// TIA Portal V15.1 export
// export: Created 2024-05-17T05:38:39.5671025Z, ExportSetting WithDefaults, DisplayName Totally Integrated Automation Portal, DisplayVersion V15.1 Update 5, DisplayName TIA Portal Openness, DisplayVersion V15.1 Update 5, DisplayName SINAMICS Startdrive Advanced, DisplayVersion V15.1, DisplayName G130, G150, S120, S150, SINAMICS MV, S210, DisplayVersion V15.1, DisplayName G110M, G120, G120C, G120D, G120P, DisplayVersion V15.1, DisplayName STEP 7 Professional, DisplayVersion V15.1 Update 5, DisplayName STEP 7 Safety, DisplayVersion V15.1, DisplayName WinCC Professional, DisplayVersion V15.1 Update 5, DisplayName SIMATIC Visualization Architect, DisplayVersion V15.1
FUNCTION_BLOCK "LGBBodyPitch"   // FB6657, FBD
TITLE = LRoller2W2S-MoviFitFCPN / LGBBodyPitch
{ S7_Optimized_Access := 'TRUE' }
AUTHOR : Imtech
FAMILY : Transport
VERSION : 0.1
// =============================================================================
// This module is used in Applications when a roller one way two speed equipped 
// with SEW MOVIFIT-FC is needed. The roller can support single body tranport and 
// simultanious transport. The roller is equipped with a standard sensor setting, 
// one stop High Speed and one at the front for dual speed transport. The 
// roller uses standard handshaking signals to accomplish an infeed transfer 
// with the previous transport system and an outfeed with the next transport 
// system.
// The roller will support automatic Mode and manual Mode according specific 
// guidelines.
// The outfeed will be master over the infeed.
// Alarm "body not in Position" is also generated.
// All Alarms coming from sub-functions, TrfIn, TrfOut & LMotor2W2S-MoviFitFCPN or 
// from 
// local Alarm are summarized to give also the global Alarm A, B, C & D to 
// upper level.
// =============================================================================
// ============================================================================
// The BodyPitch function is a local FB to be used in blowing lines transport 
// functions to handle the pitchtime between bodys.
// ============================================================================
// stored: AutoNumber false, IsIECCheckEnabled false, IsRetainMemResEnabled false, MemoryReserve 100, SetENOAutomatically False, UDAEnableTagReadback false
   VAR_INPUT
      I_PrevBodyPresentDet { ExternalAccessible := 'False'; ExternalVisible := 'False'; ExternalWritable := 'False'} : Bool;   // Previous position body present
      I_PitchDet { ExternalAccessible := 'False'; ExternalVisible := 'False'; ExternalWritable := 'False'} : Bool;   // Pitch position present
      I_ConveyorMode { ExternalAccessible := 'False'; ExternalVisible := 'False'; ExternalWritable := 'False'} : Bool;
      I_ActualPitchVal { ExternalAccessible := 'False'; ExternalVisible := 'False'; ExternalWritable := 'False'} : Int;   // Encoder pitch value in cm
      I_SkidFrontToPitchVal { ExternalAccessible := 'False'; ExternalVisible := 'False'; ExternalWritable := 'False'} : Int;   // Encoder skidfront to pitch1 value in cm
      I_PrevTransferTm { ExternalAccessible := 'False'; ExternalVisible := 'False'; ExternalWritable := 'False'} : Bool;   // Transfer previous active
      I_MotorForwardActive { ExternalAccessible := 'False'; ExternalVisible := 'False'; ExternalWritable := 'False'} : Bool;   // Motor is moving forward
      C_ConvMovFwdTime { ExternalAccessible := 'False'; ExternalVisible := 'False'; ExternalWritable := 'False'} : Time;   // Conveyor move forward time
   END_VAR
   VAR_OUTPUT
      O_BodyPitchOK { ExternalAccessible := 'False'; ExternalVisible := 'False'; ExternalWritable := 'False'} : Bool;   // Body Pitch ok
      O_ResetActualPitchVal { ExternalAccessible := 'False'; ExternalVisible := 'False'; ExternalWritable := 'False'} : Bool;   // Reset actual pitch value
      O_ResetSkidFrontToPitVal { ExternalAccessible := 'False'; ExternalVisible := 'False'; ExternalWritable := 'False'} : Bool;   // Reset skidFront to Pitch value
      O_AlarmABCondition { ExternalAccessible := 'False'; ExternalVisible := 'False'; ExternalWritable := 'False'} : Bool;   // Alarm AB Condition
      O_AlarmA { ExternalAccessible := 'False'; ExternalVisible := 'False'; ExternalWritable := 'False'} : Bool;   // Alarm A
      O_AlarmB { ExternalAccessible := 'False'; ExternalVisible := 'False'; ExternalWritable := 'False'} : Bool;   // Alarm B
      O_AlarmC { ExternalAccessible := 'False'; ExternalVisible := 'False'; ExternalWritable := 'False'} : Bool;   // Alarm C
      O_AlarmD { ExternalAccessible := 'False'; ExternalVisible := 'False'; ExternalWritable := 'False'} : Bool;   // Alarm D
   END_VAR
   VAR_IN_OUT
      IO_Modes : "Modes";   // Modes
      H_HMI : "H_HMI";   // Animation
      H_GBBodyPitch : "H_GBBodyPitch";   // Animation
   END_VAR
   VAR
      BodyPitchOK { ExternalAccessible := 'False'; ExternalVisible := 'False'; ExternalWritable := 'False'} : Bool;   // Body pitch is ok
      PitchControlWithEncoder { ExternalAccessible := 'False'; ExternalVisible := 'False'; ExternalWritable := 'False'} : Bool;   // Pitch control with encoder active
      PitchControlWithTimer { ExternalAccessible := 'False'; ExternalVisible := 'False'; ExternalWritable := 'False'} : Bool;   // Pitch control with timer active
      PitchTimeReached { ExternalAccessible := 'False'; ExternalVisible := 'False'; ExternalWritable := 'False'} : Bool;   // Pitch time is reached
      PitchDistanceReached { ExternalAccessible := 'False'; ExternalVisible := 'False'; ExternalWritable := 'False'} : Bool;   // Pitch distance is reached
      PresenceBody { ExternalAccessible := 'False'; ExternalVisible := 'False'; ExternalWritable := 'False'} : Bool;   // Body present at begin of conveyor
      AlarmA { ExternalAccessible := 'False'; ExternalVisible := 'False'; ExternalWritable := 'False'} : Bool;   // Alarm A
      AlarmB { ExternalAccessible := 'False'; ExternalVisible := 'False'; ExternalWritable := 'False'} : Bool;   // Alarm B
      AlarmC { ExternalAccessible := 'False'; ExternalVisible := 'False'; ExternalWritable := 'False'} : Bool;   // Alarm C
      AlarmD { ExternalAccessible := 'False'; ExternalVisible := 'False'; ExternalWritable := 'False'} : Bool;   // Alarm D
      AlarmABCondition { ExternalAccessible := 'False'; ExternalVisible := 'False'; ExternalWritable := 'False'} : Bool;   // Alarm AB Condition
      Edge { ExternalAccessible := 'False'; ExternalVisible := 'False'; ExternalWritable := 'False'} : Array[1..7] of Bool;   // Edge
      TimerConvMovForw { ExternalAccessible := 'False'; ExternalVisible := 'False'; ExternalWritable := 'False'} : TOF_TIME;   // Timer
      PitchTimer { ExternalAccessible := 'False'; ExternalVisible := 'False'; ExternalWritable := 'False'} : "LTimer";   // Pitch Timer
   END_VAR
   VAR_TEMP
      HMICMD : Struct   // Temp
         PitchControlWithTimerSel : Bool;   // Pitch control with timer selected
         PitchControlWithEncoderSel : Bool;   // Pitch control with encoder selected
         Spare2 : Bool;   // Spare
         Spare3 : Bool;   // Spare
         Spare4 : Bool;   // Spare
         Spare5 : Bool;   // Spare
         Spare6 : Bool;   // Spare
         Spare7 : Bool;   // Spare
         Spare8 : Bool;   // Spare
         Spare9 : Bool;   // Spare
         Spare10 : Bool;   // Spare
         Spare11 : Bool;   // Spare
         Spare12 : Bool;   // Spare
         Spare13 : Bool;   // Spare
         Spare14 : Bool;   // Spare
         Spare15 : Bool;   // Spare
         Spare16 : Bool;   // Spare
         Spare17 : Bool;   // Spare
         Spare18 : Bool;   // Spare
         Spare19 : Bool;   // Spare
         Spare20 : Bool;   // Spare
         Spare21 : Bool;   // Spare
         Spare22 : Bool;   // Spare
         Spare23 : Bool;   // Spare
         Spare24 : Bool;   // Spare
         Spare25 : Bool;   // Spare
         Spare26 : Bool;   // Spare
         Spare27 : Bool;   // Spare
         Spare28 : Bool;   // Spare
         Spare29 : Bool;   // Spare
         Spare30 : Bool;   // Spare
         Spare31 : Bool;   // Spare
      END_STRUCT;
      TempInt : Int;   // Temp
      TempDInt : DInt;   // Temp / Temp DInt
      TempReal : Real;   // Temp
   END_VAR
   VAR_TEMP   // added for the SCL form of the ladder/FBD networks
      _w1 : Bool;
      _w2 : Bool;
   END_VAR
BEGIN

REGION Network 1: **** 1 - Inputs **** HMI Commands
   // HMI Commands
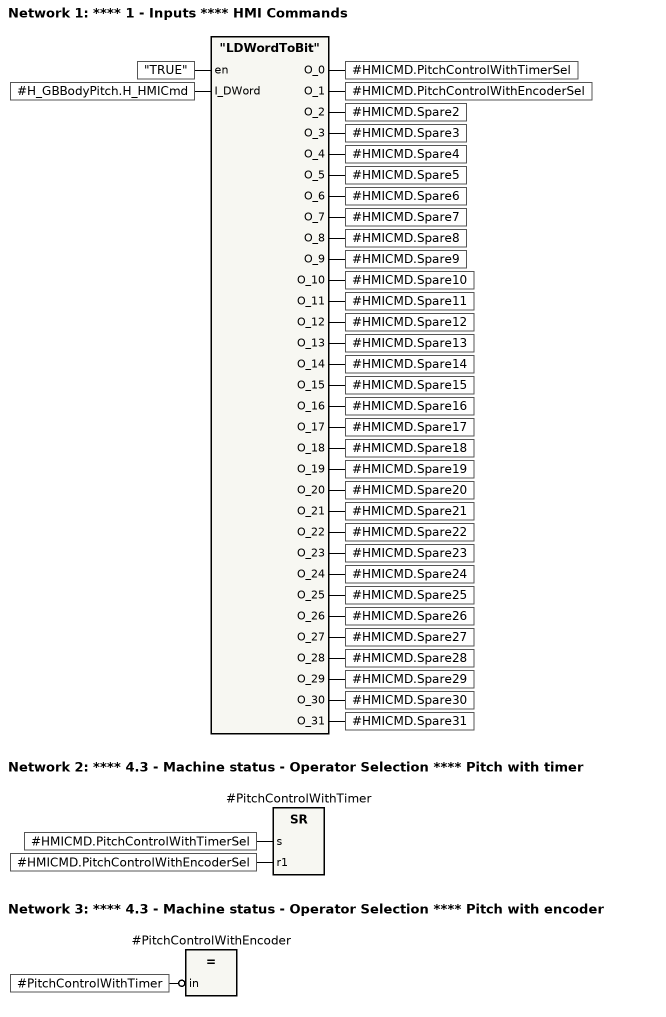
   IF "TRUE" THEN
       "LDWordToBit"(I_DWord := #H_GBBodyPitch.H_HMICmd,
                     O_0 => #HMICMD.PitchControlWithTimerSel,
                     O_1 => #HMICMD.PitchControlWithEncoderSel,
                     O_2 => #HMICMD.Spare2,
                     O_3 => #HMICMD.Spare3,
                     O_4 => #HMICMD.Spare4,
                     O_5 => #HMICMD.Spare5,
                     O_6 => #HMICMD.Spare6,
                     O_7 => #HMICMD.Spare7,
                     O_8 => #HMICMD.Spare8,
                     O_9 => #HMICMD.Spare9,
                     O_10 => #HMICMD.Spare10,
                     O_11 => #HMICMD.Spare11,
                     O_12 => #HMICMD.Spare12,
                     O_13 => #HMICMD.Spare13,
                     O_14 => #HMICMD.Spare14,
                     O_15 => #HMICMD.Spare15,
                     O_16 => #HMICMD.Spare16,
                     O_17 => #HMICMD.Spare17,
                     O_18 => #HMICMD.Spare18,
                     O_19 => #HMICMD.Spare19,
                     O_20 => #HMICMD.Spare20,
                     O_21 => #HMICMD.Spare21,
                     O_22 => #HMICMD.Spare22,
                     O_23 => #HMICMD.Spare23,
                     O_24 => #HMICMD.Spare24,
                     O_25 => #HMICMD.Spare25,
                     O_26 => #HMICMD.Spare26,
                     O_27 => #HMICMD.Spare27,
                     O_28 => #HMICMD.Spare28,
                     O_29 => #HMICMD.Spare29,
                     O_30 => #HMICMD.Spare30,
                     O_31 => #HMICMD.Spare31);
   END_IF;
END_REGION

REGION Network 2: **** 4.3 - Machine status - Operator Selection **** Pitch with timer
   IF #HMICMD.PitchControlWithTimerSel THEN
       #PitchControlWithTimer := TRUE;   // SR flip-flop
   END_IF;
   IF #HMICMD.PitchControlWithEncoderSel THEN #PitchControlWithTimer := FALSE; END_IF;
END_REGION

REGION Network 3: **** 4.3 - Machine status - Operator Selection **** Pitch with encoder
   #PitchControlWithEncoder := NOT #PitchControlWithTimer;
END_REGION

REGION Network 4: **** 4.4 - Machine status - Calculated **** Logger skidfront - pitch sensor distance
   // Simple logger for skidfront - pitch sensor distance
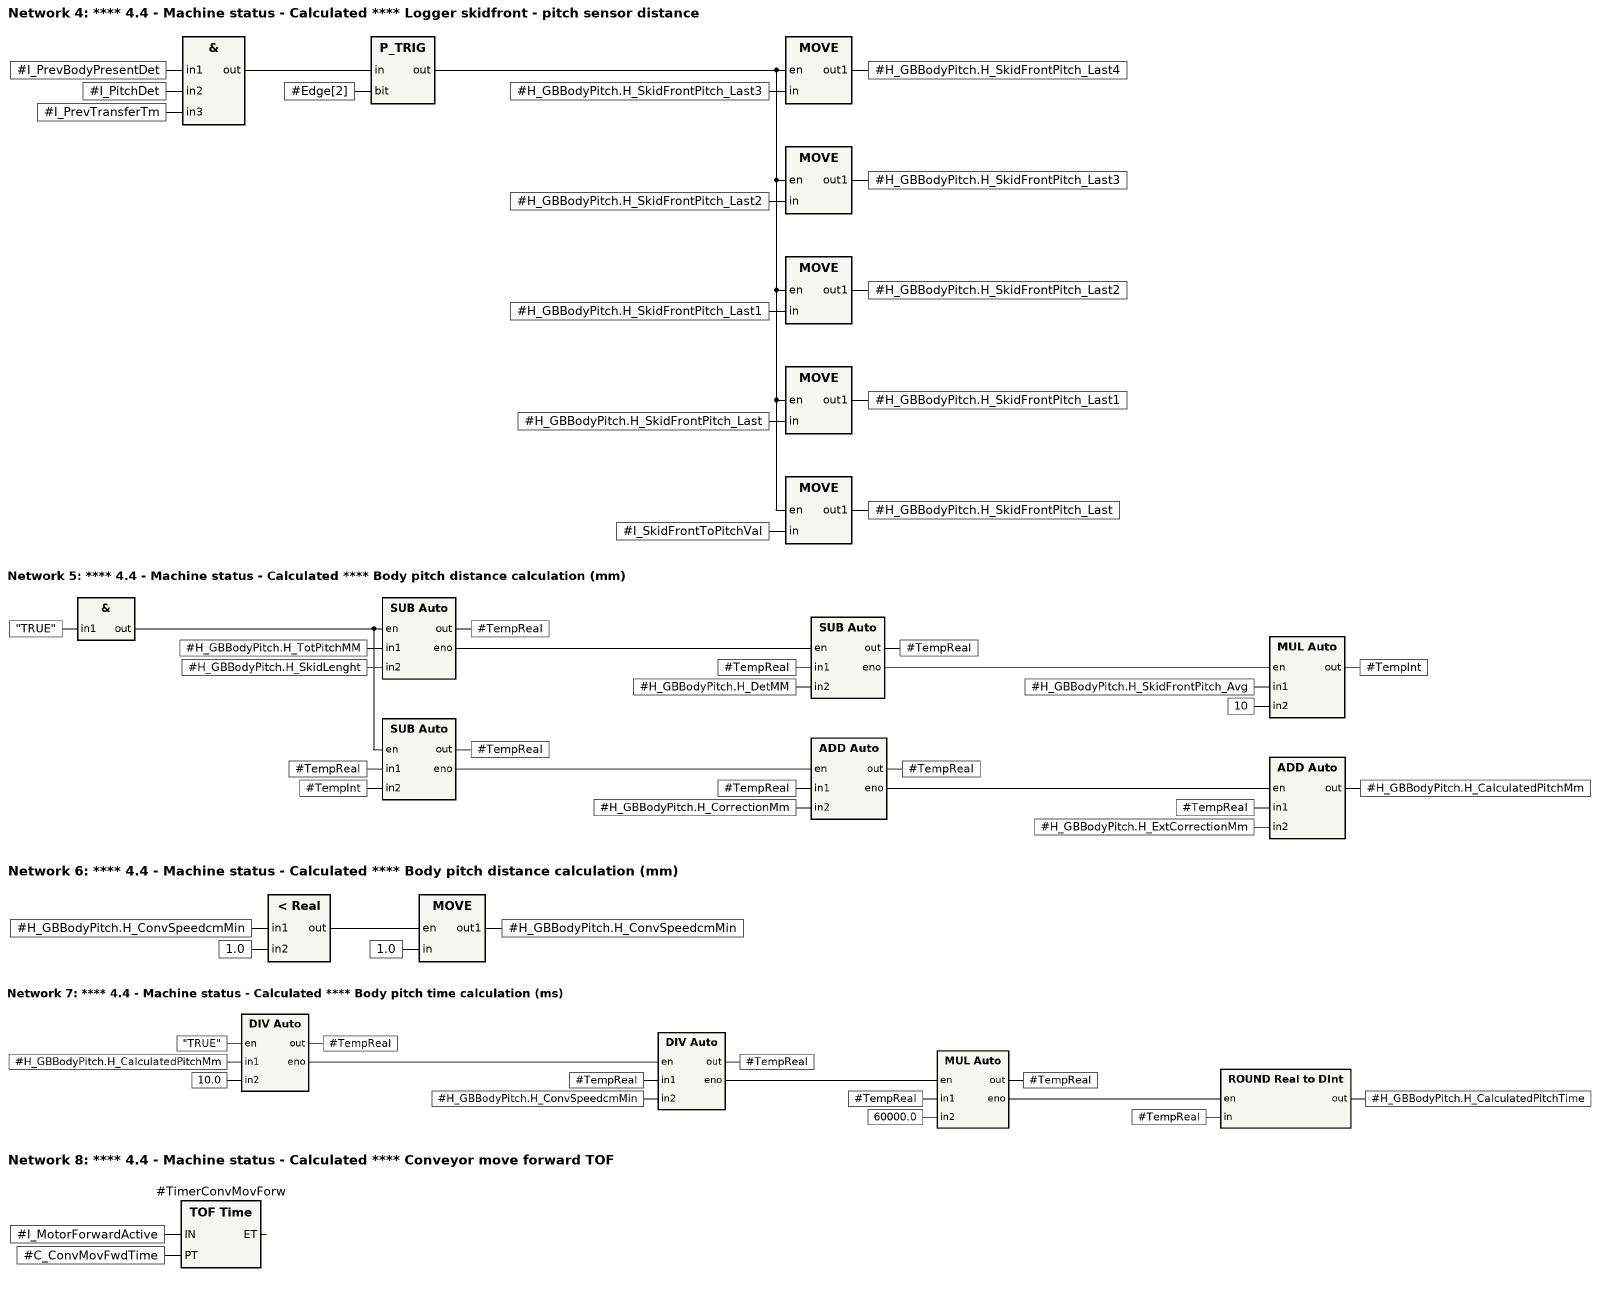
   #_w1 := #I_PrevBodyPresentDet AND #I_PitchDet AND #I_PrevTransferTm;
   #_w2 := #_w1 AND NOT #Edge[2];   // rising edge
   #Edge[2] := #_w1;
   IF #_w2 THEN
       #H_GBBodyPitch.H_SkidFrontPitch_Last4 := #H_GBBodyPitch.H_SkidFrontPitch_Last3;
       #H_GBBodyPitch.H_SkidFrontPitch_Last3 := #H_GBBodyPitch.H_SkidFrontPitch_Last2;
       #H_GBBodyPitch.H_SkidFrontPitch_Last2 := #H_GBBodyPitch.H_SkidFrontPitch_Last1;
       #H_GBBodyPitch.H_SkidFrontPitch_Last1 := #H_GBBodyPitch.H_SkidFrontPitch_Last;
       #H_GBBodyPitch.H_SkidFrontPitch_Last := #I_SkidFrontToPitchVal;
   END_IF;
END_REGION

REGION Network 5: **** 4.4 - Machine status - Calculated **** Body pitch distance calculation (mm)
   IF "TRUE" THEN
       #TempReal := #H_GBBodyPitch.H_TotPitchMM - #H_GBBodyPitch.H_SkidLenght;
       #TempReal := #TempReal - #H_GBBodyPitch.H_DetMM;
       #TempInt := #H_GBBodyPitch.H_SkidFrontPitch_Avg * 10;
       #TempReal := #TempReal - #TempInt;
       #TempReal := #TempReal + #H_GBBodyPitch.H_CorrectionMm;
       #H_GBBodyPitch.H_CalculatedPitchMm := #TempReal + #H_GBBodyPitch.H_ExtCorrectionMm;
   END_IF;
END_REGION

REGION Network 6: **** 4.4 - Machine status - Calculated **** Body pitch distance calculation (mm)
   // Prevent to devide by zero at the body pitch time calculation network
   IF #H_GBBodyPitch.H_ConvSpeedcmMin < 1.0 THEN #H_GBBodyPitch.H_ConvSpeedcmMin := 1.0; END_IF;
END_REGION

REGION Network 7: **** 4.4 - Machine status - Calculated **** Body pitch time calculation (ms)
   IF "TRUE" THEN
       #TempReal := #H_GBBodyPitch.H_CalculatedPitchMm / 10.0;
       #TempReal := #TempReal / #H_GBBodyPitch.H_ConvSpeedcmMin;
       #TempReal := #TempReal * 60000.0;
       #H_GBBodyPitch.H_CalculatedPitchTime := ROUND(#TempReal);
   END_IF;
END_REGION

REGION Network 8: **** 4.4 - Machine status - Calculated **** Conveyor move forward TOF
   #TimerConvMovForw(IN := #I_MotorForwardActive, PT := #C_ConvMovFwdTime);   // TOF
END_REGION

REGION Network 9: **** 4.4 - Machine status - Calculated **** Pitch timer
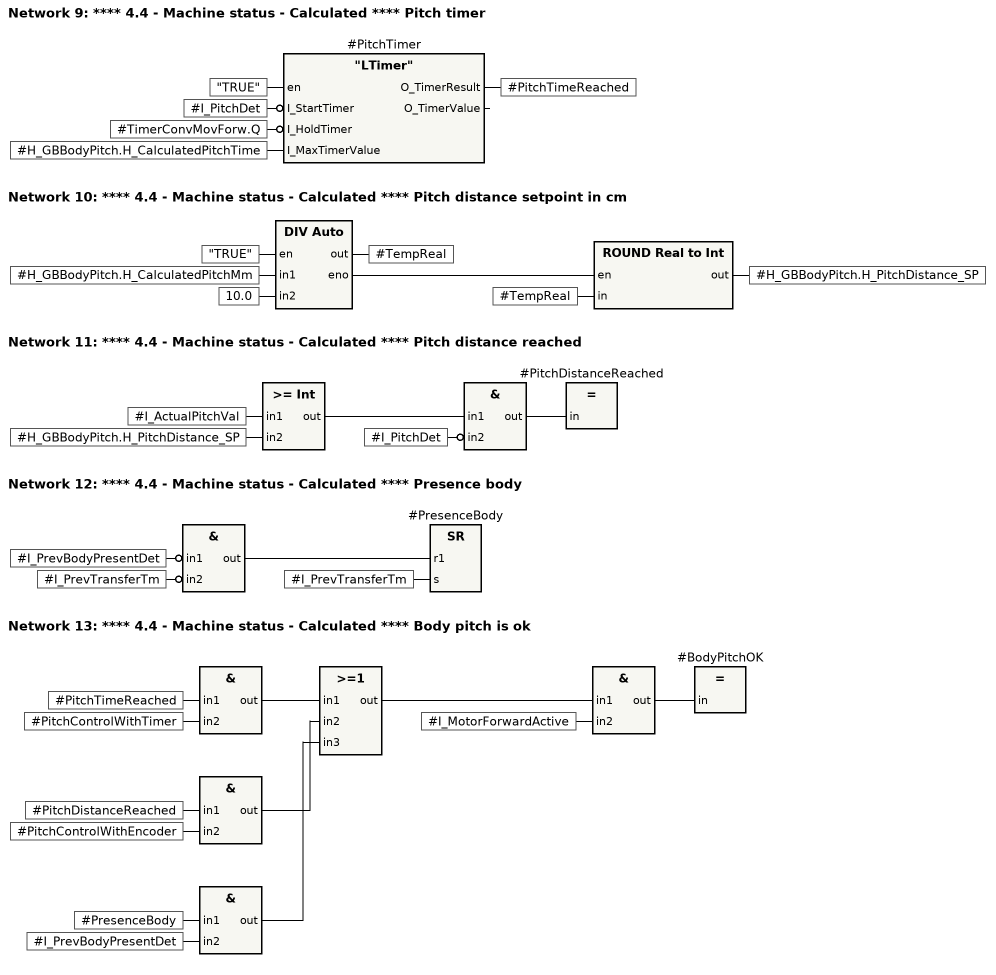
   IF "TRUE" THEN
       #PitchTimer(I_StartTimer := NOT #I_PitchDet,   // "LTimer"
                   I_HoldTimer := NOT #TimerConvMovForw.Q,
                   I_MaxTimerValue := #H_GBBodyPitch.H_CalculatedPitchTime,
                   O_TimerResult => #PitchTimeReached);
   END_IF;
END_REGION

REGION Network 10: **** 4.4 - Machine status - Calculated **** Pitch distance setpoint in cm
   IF "TRUE" THEN
       #TempReal := #H_GBBodyPitch.H_CalculatedPitchMm / 10.0;
       #H_GBBodyPitch.H_PitchDistance_SP := ROUND(#TempReal);
   END_IF;
END_REGION

REGION Network 11: **** 4.4 - Machine status - Calculated **** Pitch distance reached
   #PitchDistanceReached := (#I_ActualPitchVal >= #H_GBBodyPitch.H_PitchDistance_SP) AND NOT #I_PitchDet;
END_REGION

REGION Network 12: **** 4.4 - Machine status - Calculated **** Presence body
   // Presence body at begin of conveyor
   IF #I_PrevTransferTm THEN
       #PresenceBody := TRUE;   // SR flip-flop
   END_IF;
   IF NOT #I_PrevBodyPresentDet AND NOT #I_PrevTransferTm THEN #PresenceBody := FALSE; END_IF;
END_REGION

REGION Network 13: **** 4.4 - Machine status - Calculated **** Body pitch is ok
   #BodyPitchOK := ((#PitchTimeReached AND #PitchControlWithTimer) OR (#PitchDistanceReached AND #PitchControlWithEncoder) OR (#PresenceBody AND #I_PrevBodyPresentDet)) AND #I_MotorForwardActive;
END_REGION

REGION Network 14: **** 4.6 - Machine Status - Indication **** Icon Animation
   // Icon Animation
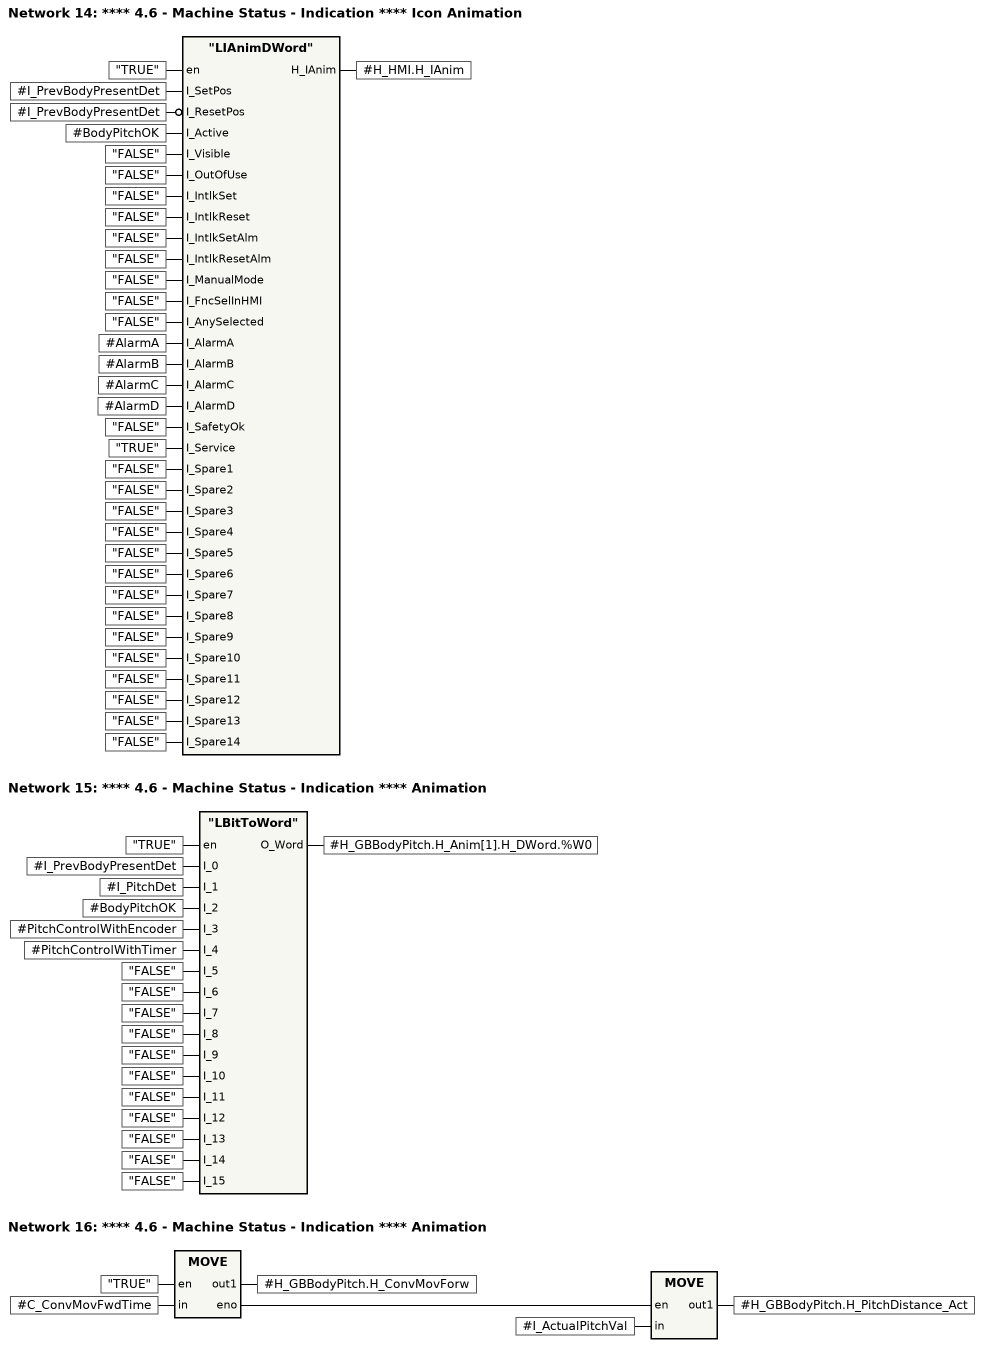
   IF "TRUE" THEN
       "LIAnimDWord"(I_SetPos := #I_PrevBodyPresentDet,
                     I_ResetPos := NOT #I_PrevBodyPresentDet,
                     I_Active := #BodyPitchOK,
                     I_Visible := "FALSE",
                     I_OutOfUse := "FALSE",
                     I_IntlkSet := "FALSE",
                     I_IntlkReset := "FALSE",
                     I_IntlkSetAlm := "FALSE",
                     I_IntlkResetAlm := "FALSE",
                     I_ManualMode := "FALSE",
                     I_FncSelInHMI := "FALSE",
                     I_AnySelected := "FALSE",
                     I_AlarmA := #AlarmA,
                     I_AlarmB := #AlarmB,
                     I_AlarmC := #AlarmC,
                     I_AlarmD := #AlarmD,
                     I_SafetyOk := "FALSE",
                     I_Service := "TRUE",
                     I_Spare1 := "FALSE",
                     I_Spare2 := "FALSE",
                     I_Spare3 := "FALSE",
                     I_Spare4 := "FALSE",
                     I_Spare5 := "FALSE",
                     I_Spare6 := "FALSE",
                     I_Spare7 := "FALSE",
                     I_Spare8 := "FALSE",
                     I_Spare9 := "FALSE",
                     I_Spare10 := "FALSE",
                     I_Spare11 := "FALSE",
                     I_Spare12 := "FALSE",
                     I_Spare13 := "FALSE",
                     I_Spare14 := "FALSE",
                     H_IAnim => #H_HMI.H_IAnim);
   END_IF;
END_REGION

REGION Network 15: **** 4.6 - Machine Status - Indication **** Animation
   // Animation
   IF "TRUE" THEN
       "LBitToWord"(I_0 := #I_PrevBodyPresentDet,
                    I_1 := #I_PitchDet,
                    I_2 := #BodyPitchOK,
                    I_3 := #PitchControlWithEncoder,
                    I_4 := #PitchControlWithTimer,
                    I_5 := "FALSE",
                    I_6 := "FALSE",
                    I_7 := "FALSE",
                    I_8 := "FALSE",
                    I_9 := "FALSE",
                    I_10 := "FALSE",
                    I_11 := "FALSE",
                    I_12 := "FALSE",
                    I_13 := "FALSE",
                    I_14 := "FALSE",
                    I_15 := "FALSE",
                    O_Word => #H_GBBodyPitch.H_Anim[1].H_DWord.%W0);
   END_IF;
END_REGION

REGION Network 16: **** 4.6 - Machine Status - Indication **** Animation
   IF "TRUE" THEN
       #H_GBBodyPitch.H_ConvMovForw := #C_ConvMovFwdTime;
       #H_GBBodyPitch.H_PitchDistance_Act := #I_ActualPitchVal;
   END_IF;
END_REGION

REGION Network 17: **** 8 - Outputs **** Reset Actual Pitch value
   // Pitch counter (with encoder)
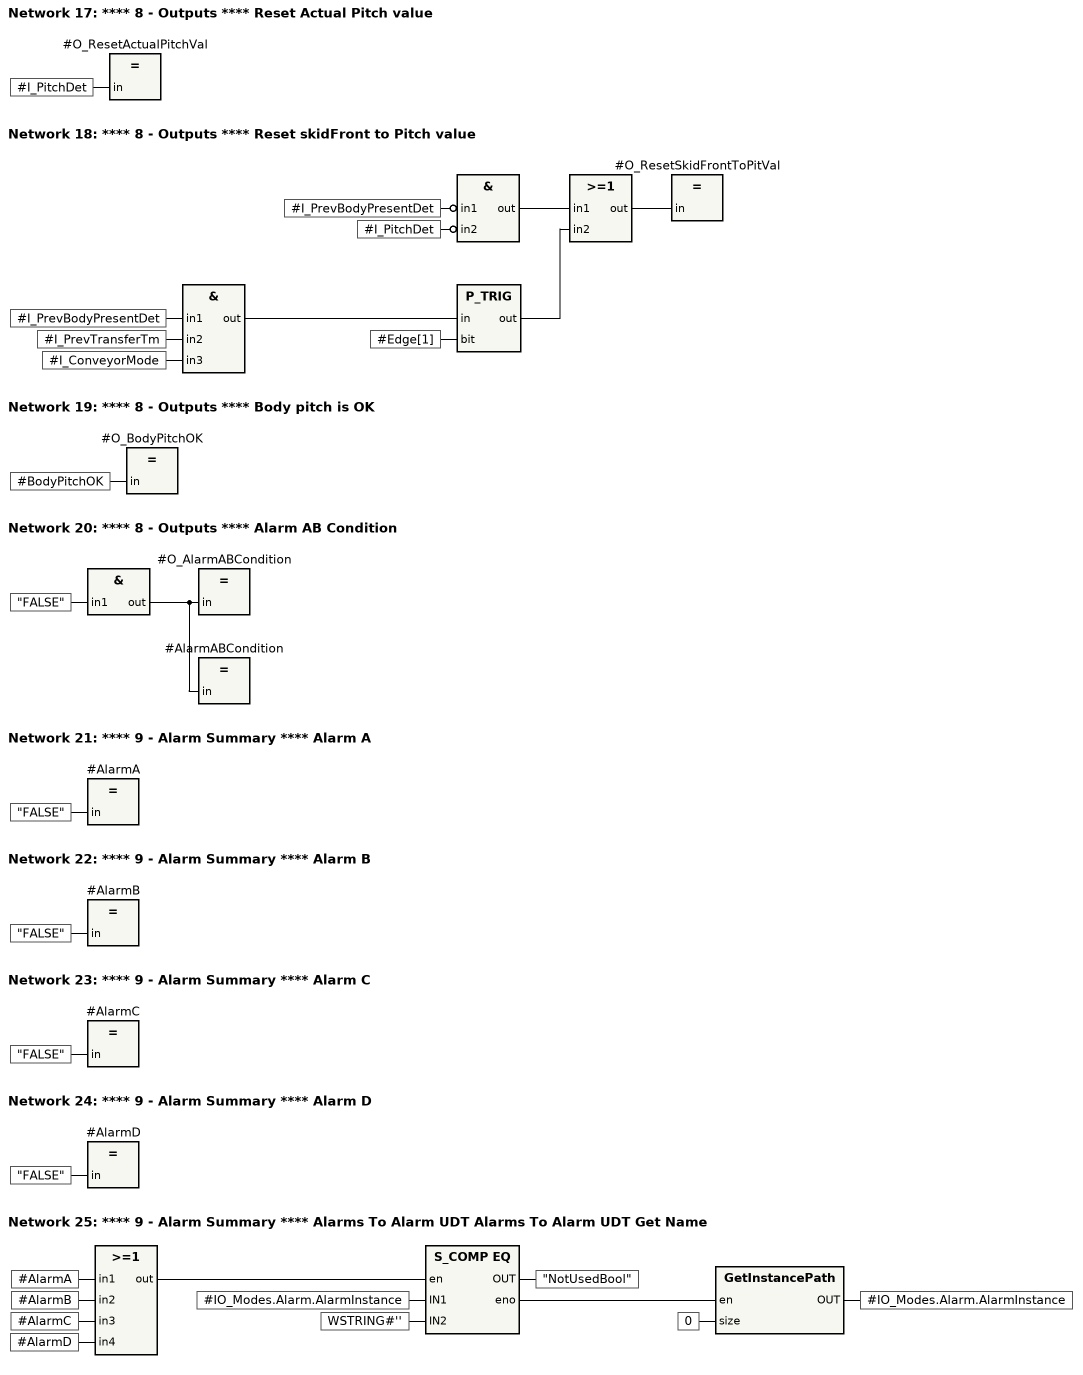
   #O_ResetActualPitchVal := #I_PitchDet;
END_REGION

REGION Network 18: **** 8 - Outputs **** Reset skidFront to Pitch value
   // Reset the skidfront to pitch value (No body between PrevBody det and Pitch 
   // det), what is the distance between the 2 sensors. The input PrevTransfetTM is 
   // set when the trf start from Prev to next.
   #_w1 := #I_PrevBodyPresentDet AND #I_PrevTransferTm AND #I_ConveyorMode;
   #_w2 := #_w1 AND NOT #Edge[1];   // rising edge
   #Edge[1] := #_w1;
   #O_ResetSkidFrontToPitVal := (NOT #I_PrevBodyPresentDet AND NOT #I_PitchDet) OR #_w2;
END_REGION

REGION Network 19: **** 8 - Outputs **** Body pitch is OK
   #O_BodyPitchOK := #BodyPitchOK;
END_REGION

REGION Network 20: **** 8 - Outputs **** Alarm AB Condition
   // Alarm AB Condition
   #O_AlarmABCondition := "FALSE";
   #AlarmABCondition := "FALSE";
END_REGION

REGION Network 21: **** 9 - Alarm Summary **** Alarm A
   // Alarms A
   #AlarmA := "FALSE";
END_REGION

REGION Network 22: **** 9 - Alarm Summary **** Alarm B
   // Alarms B
   #AlarmB := "FALSE";
END_REGION

REGION Network 23: **** 9 - Alarm Summary **** Alarm C
   // Alarms C
   #AlarmC := "FALSE";
END_REGION

REGION Network 24: **** 9 - Alarm Summary **** Alarm D
   // Alarms D
   #AlarmD := "FALSE";
END_REGION

REGION Network 25: **** 9 - Alarm Summary **** Alarms To Alarm UDT Alarms To Alarm UDT Get Name
   // Alarm D
   S_COMP(EN := #AlarmA OR #AlarmB OR #AlarmC OR #AlarmD,
          IN1 := #IO_Modes.Alarm.AlarmInstance,
          IN2 := WSTRING#'',
          OUT => "NotUsedBool",
          ENO => #_w1);
   IF #_w1 THEN GetInstancePath(size := 0, OUT => #IO_Modes.Alarm.AlarmInstance); END_IF;
END_REGION

REGION Network 26: **** 9 - Alarm Summary **** Alarms To Alarm UDT
   // Alarm D
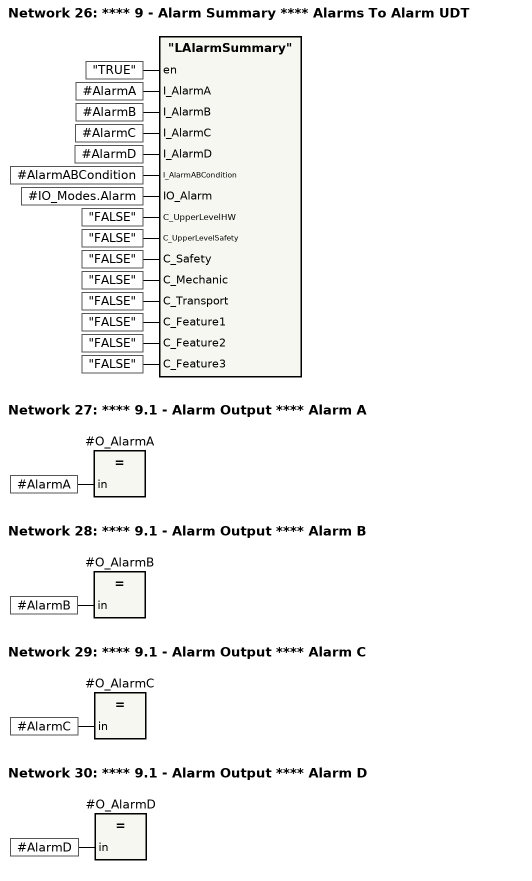
   IF "TRUE" THEN
       "LAlarmSummary"(I_AlarmA := #AlarmA,
                       I_AlarmB := #AlarmB,
                       I_AlarmC := #AlarmC,
                       I_AlarmD := #AlarmD,
                       I_AlarmABCondition := #AlarmABCondition,
                       IO_Alarm := #IO_Modes.Alarm,
                       C_UpperLevelHW := "FALSE",
                       C_UpperLevelSafety := "FALSE",
                       C_Safety := "FALSE",
                       C_Mechanic := "FALSE",
                       C_Transport := "FALSE",
                       C_Feature1 := "FALSE",
                       C_Feature2 := "FALSE",
                       C_Feature3 := "FALSE");
   END_IF;
END_REGION

REGION Network 27: **** 9.1 - Alarm Output **** Alarm A
   // Alarms A
   #O_AlarmA := #AlarmA;
END_REGION

REGION Network 28: **** 9.1 - Alarm Output **** Alarm B
   // Alarms B
   #O_AlarmB := #AlarmB;
END_REGION

REGION Network 29: **** 9.1 - Alarm Output **** Alarm C
   // Alarms C
   #O_AlarmC := #AlarmC;
END_REGION

REGION Network 30: **** 9.1 - Alarm Output **** Alarm D
   // Alarms D
   #O_AlarmD := #AlarmD;
END_REGION
END_FUNCTION_BLOCK
